// TIA Portal V16 export
// export: Created 2024-09-05T17:39:24.5402005Z, ExportSetting WithDefaults, DisplayName Totally Integrated Automation Portal, DisplayVersion V16 Update 6, DisplayName TIA Portal Version Control Interface, DisplayVersion V16 Update 2, DisplayName TIA Portal Openness, DisplayVersion V16 Update 6, DisplayName STEP 7 Professional, DisplayVersion V16 Update 6, DisplayName STEP 7 Safety, DisplayVersion V16, DisplayName WinCC Advanced, DisplayVersion V16 Update 6
FUNCTION "FC_DMC" : Void   // FC2012, LAD
{ S7_Optimized_Access := 'TRUE' }
VERSION : 0.1
// stored: AutoNumber false, IsIECCheckEnabled false, SetENOAutomatically false, UDAEnableTagReadback false
   VAR_TEMP
      stationName1 : WString;
      stationName2 : WString;
      Data_DMC : Array[1.."MaxRoundNumber", 1..10] of "DATA_DMC";
      timeUTC : DTL;
      _ret_val : Int;
   END_VAR
BEGIN

REGION Network 1
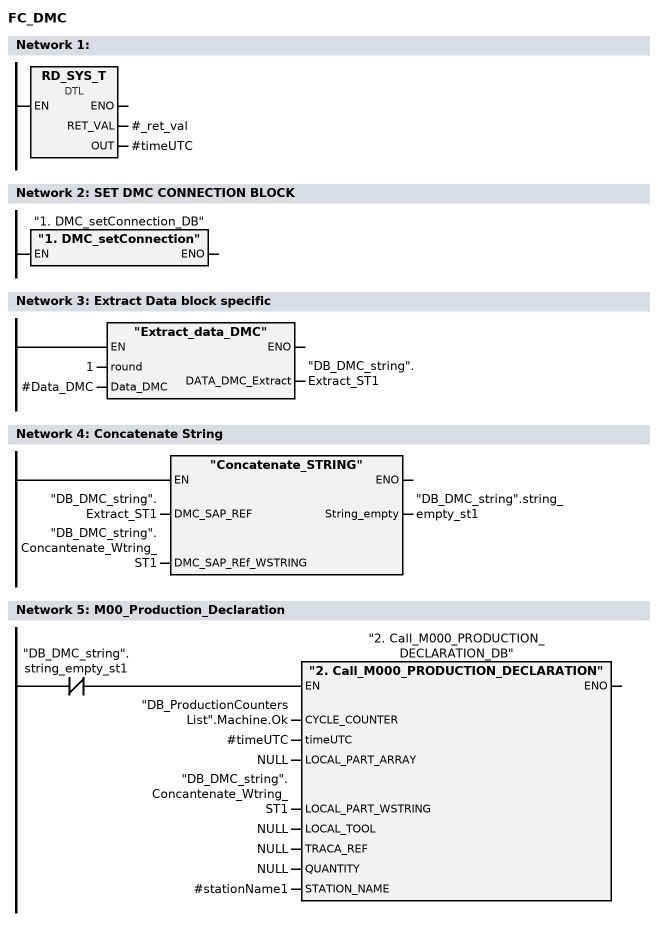
   RUNG wire#powerrail
      { S7_Templates := "date_type := DTL" } RD_SYS_T(RET_VAL => #_ret_val, OUT => #timeUTC)
   END_RUNG
   // the same network as SCL:
   #_ret_val := RD_SYS_T(OUT => #timeUTC);
END_REGION

REGION Network 2: SET DMC CONNECTION BLOCK
   RUNG wire#powerrail
      "1. DMC_setConnection_DB"()
   END_RUNG
   // the same network as SCL:
   "1. DMC_setConnection_DB"();   // "1. DMC_setConnection"
END_REGION

REGION Network 3: Extract Data block specific
   RUNG wire#powerrail
      "Extract_data_DMC"(round := 1, Data_DMC := #Data_DMC, DATA_DMC_Extract => "DB_DMC_string".Extract_ST1)
   END_RUNG
   // the same network as SCL:
   "Extract_data_DMC"(round := 1, Data_DMC := #Data_DMC, DATA_DMC_Extract => "DB_DMC_string".Extract_ST1);
END_REGION

REGION Network 4: Concatenate String
   RUNG wire#powerrail
      "Concatenate_STRING"(DMC_SAP_REF := "DB_DMC_string".Extract_ST1, DMC_SAP_REf_WSTRING := "DB_DMC_string".Concantenate_Wtring_ST1, String_empty => "DB_DMC_string".string_empty_st1)
   END_RUNG
   // the same network as SCL:
   "Concatenate_STRING"(DMC_SAP_REF := "DB_DMC_string".Extract_ST1,
                        DMC_SAP_REf_WSTRING := "DB_DMC_string".Concantenate_Wtring_ST1,
                        String_empty => "DB_DMC_string".string_empty_st1);
END_REGION

REGION Network 5: M00_Production_Declaration
   RUNG wire#powerrail
      I_Contact( "DB_DMC_string".string_empty_st1 )
      "2. Call_M000_PRODUCTION_DECLARATION_DB"(CYCLE_COUNTER := "DB_ProductionCountersList".Machine.Ok, timeUTC := #timeUTC, LOCAL_PART_ARRAY := NULL, LOCAL_PART_WSTRING := "DB_DMC_string".Concantenate_Wtring_ST1, LOCAL_TOOL := NULL, TRACA_REF := NULL, QUANTITY := NULL, STATION_NAME := #stationName1)
   END_RUNG
   // the same network as SCL:
   IF NOT "DB_DMC_string".string_empty_st1 THEN
       "2. Call_M000_PRODUCTION_DECLARATION_DB"(CYCLE_COUNTER := "DB_ProductionCountersList".Machine.Ok,   // "2. Call_M000_PRODUCTION_DECLARATION"
                               timeUTC := #timeUTC,
                               LOCAL_PART_ARRAY := NULL,
                               LOCAL_PART_WSTRING := "DB_DMC_string".Concantenate_Wtring_ST1,
                               LOCAL_TOOL := NULL,
                               TRACA_REF := NULL,
                               QUANTITY := NULL,
                               STATION_NAME := #stationName1);
   END_IF;
END_REGION
END_FUNCTION
